(* www.hevs.ch Institut Systemes Industriels Project: HEVS Pack 2022 Author: Cedric Lenoir Date: 2024 August 30 This Function Block compute time statistics *)
FUNCTION_BLOCK FB_PackStatistic
  VAR_INPUT
    Enable : BOOL;
  END_VAR
  VAR_IN_OUT
    plcCurrentTime_s : UDINT;  (* E.g from PackTag.hevsPackTime.Local_date_time_seconds *)
    unitCurrentMode : E_PackModes;
    unitCurrentState : E_PackState;
    unitAdmin : HEVS_PackTag_Admin;
  END_VAR
  VAR_OUTPUT
    Active : BOOL;
  END_VAR
  VAR
    trigModeTimeCurrent : R_TRIG;  (* Detext State / Mode change *)
    trigStateTimeCurrent : R_TRIG;
    memCurrentMode : E_PackModes := E_PackModes.Invalid;
    memCurrentState : E_PackState := E_PackState.eUndefined;
    timeModeAtTrigger_s : UDINT;  (* Start time at trigger to compute current *)
    timeStateAtTrigger_s : UDINT;
    bProgramStarted : BOOL;
    timeProgramStarted_s : UDINT;
    getMemCumTimeMode : DINT;  (* Get Time In CumulativeTime for Mode and or state *)
    getMemCumTimeModeState : DINT;
  END_VAR

                  IF Enable THEN
	trigModeTimeCurrent(clk := (unitCurrentMode <> memCurrentMode));
	trigStateTimeCurrent(clk := (unitCurrentState <> memCurrentState));
	
	IF trigModeTimeCurrent.Q THEN
		timeModeAtTrigger_s := plcCurrentTime_s;
		memCurrentMode := unitCurrentMode;
		// Get Stored value to compute new cummulative time.
		getMemCumTimeMode := unitAdmin.CumulativeTime[0].ModeStateTimes[unitCurrentMode].Mode;
	END_IF
	
	IF trigStateTimeCurrent.Q THEN
		timeStateAtTrigger_s := plcCurrentTime_s;
		memCurrentState := unitCurrentState;
	END_IF
	
	// If mode or state changed
	IF trigModeTimeCurrent.Q  OR
	   trigStateTimeCurrent.Q THEN
	   getMemCumTimeModeState := unitAdmin.CumulativeTime[0].ModeStateTimes[unitCurrentMode].State[memCurrentState];
	END_IF
	
	IF NOT bProgramStarted THEN
		bProgramStarted := TRUE;
		timeProgramStarted_s := plcCurrentTime_s;
	END_IF
	
	unitAdmin.ModeTimeCurrent := UDINT_TO_DINT(plcCurrentTime_s - timeModeAtTrigger_s);
	
	unitAdmin.StateTimeCurrent := UDINT_TO_DINT(plcCurrentTime_s - timeStateAtTrigger_s);
	
	// Default for [*] time from start program
	// No retain, that is number of Sec since last restart.
	unitAdmin.CumulativeTime[0].AccTimeSinceReset := UDINT_TO_DINT(plcCurrentTime_s - timeProgramStarted_s);
	
	// Minimum protection in case of unitCurrentMode exceed 
	//	HEVS_PackTag_GVL.C_MAXMODSTATESTIMES
	IF unitCurrentMode <= HEVS_PackTag_GVL.C_MAXMODSTATESTIMES THEN
		// getMemCumTimeMode is set only at trigger change mode
		unitAdmin.CumulativeTime[0].ModeStateTimes[unitCurrentMode].Mode := getMemCumTimeMode + unitAdmin.ModeTimeCurrent;
	END_IF
	
	// Minimum protection in case of unitCurrentMode exceed 
	//	HEVS_PackTag_GVL.C_MAXMODSTATESTIMES
	// 	HEVS_PackTag_GVL.C_MAXSTATES
	IF unitCurrentMode <= HEVS_PackTag_GVL.C_MAXMODSTATESTIMES AND
	   unitCurrentState <= HEVS_PackTag_GVL.C_MAXSTATES        THEN
		// getMemCumTimeModeState is set only at trigger change of mode OR state 
		unitAdmin.CumulativeTime[0].ModeStateTimes[unitCurrentMode].State[unitCurrentState] := getMemCumTimeModeState +  unitAdmin.StateTimeCurrent;
	END_IF
	
	Active	:= FALSE;
ELSE
	
	Active	:= TRUE;
END_IF




                
END_FUNCTION_BLOCK

CONFIGURATION Application
  RESOURCE Application ON PLC
    {attribute 'qualified_only'}
    VAR_GLOBAL CONSTANT  (* HEVS_PackTag_GVL - List of PackTags based on ISA–TR88.00.02-2022 www.hevs.ch Institut Systemes Industriels / Power & Control Project: Automation Box CtrlX S3 Author: Romain Ferrari & Cedric Lenoir Date: 2024 July 31 !!!!!! The value of these constants have to be set by the user depending on the system it is implemented on. !!!!!!\\ *)
      C_MAXSTATES : INT := 17;  (* Max State number. 0 is invalid *)
      C_COMMAND_MAXREALPARAMS : INT := 8;
      C_COMMAND_MAXSTRINGPARAMS : INT := 2;  (* / *)
      C_COMMAND_MAXLREALPARAMS : INT := 8;  (* Used in one of the main PackTag branch of the HEVS_PackTag_V30 : Command *)
      C_COMMAND_MAXDINTPARAMS : INT := 8;
      C_COMMAND_MAXRECIPE : INT := 8;
      C_STATUS_MAXREALPARAMS : INT := 8;  (* / *)
      C_STATUS_MAXSTRINGPARAMS : INT := 2;  (* / *)
      C_STATUS_MAXLREALPARAMS : INT := 8;
      C_STATUS_MAXDINTPARAMS : INT := 8;  (* Used in one of the main PackTag branch of the HEVS_PackTag_V30 : Status *)
      C_STATUS_MAXRECIPE : INT := 8;
      C_STATUS_MAXSTACKLIGHT : INT := 8;
      C_ADMIN_MAXREALPARAMS : INT := 8;  (* / *)
      C_ADMIN_MAXSTRINGPARAMS : INT := 2;  (* / *)
      C_ADMIN_MAXLREALPARAMS : INT := 8;
      C_ADMIN_MAXDINTPARAMS : INT := 8;
      C_ADMIN_MAXALARMS : INT := 20;
      C_ADMIN_MAXHISTORYALARMS : INT := 20;
      C_ADMIN_MAXWARNINGS : INT := 20;
      C_ADMIN_MAXCUMULATIVETIMES : INT := 3;  (* Minimum is 0 for [0], Arbitrarily initialized to 3 *)
      C_ADMIN_MAXPRODUCTDATA : INT := 11;
      C_ADMIN_MAXDISABLEDSTATES : INT := 8;
      C_ADMIN_MAXMODESTRANSITION : INT := 8;  (* is absolutely limited by C_ADMIN_MAXMODESTRANSITIONPACK *)
      C_ADMIN_MAXMODESTRANSITIONPACK : INT := 31;  (* as Pack used DWORD and 0 is reserved, max is limited to 31 *)
      C_MAXMODSTATESTIMES : INT := 8;
      C_MAXREALVARIABLES : INT := 8;
      C_MAXSTRINGVARIABLES : INT := 8;
      C_MAXLREALVARIABLES : INT := 8;
      C_MAXDINTVARIABLES : INT := 8;  (* Used in lower branches of the HEVS_PackTag_V30 *)
      C_MAXREALINGREDIENTS : INT := 8;
      C_MAXSTRINGINGREDIENTS : INT := 8;
      C_MAXLREALINGREDIENTS : INT := 8;
      C_MAXDINTINGREDIENTS : INT := 8;
      hevs_min_packtag_v2022 : HEVS_Min_PackTag_V2022;
    END_VAR
    {attribute 'qualified_only'}
    VAR_GLOBAL  (* PackTag - www.hevs.ch Institut Systemes Industriels Project: HEVS Pack 2022 Author: Cedric Lenoir Date: 2024 August 29 Base GVL for HEVS Pack Tag File name should be PackTag *)
      Command : HEVS_PackTag_Command;
      Status : HEVS_PackTag_Status;
      Admin : HEVS_PackTag_Admin;
      hevsPackTime : HEVS_Time;  (* HEVS Time, needed for Alarms and Time in Pack Computed with PRG_GetTime_CtrlX or PRG_GetTime_TwinCAT or Your own system *)
      hevsUI : HEVS_PackTag_UI;  (* Help for interface and diagnostic HEVS Pack could be used without this Struct. Can be used with fbCmdBoolInterface Can be used with fbGetActualBoolState *)
      hevsPackAlarm_UI : HEVS_PackAlarm_UI;  (* Help for interface and diagnostic HEVS Pack could be used without this Struct. Can be used with program PRG_TestAlarm *)
    END_VAR
    {attribute 'qualified_only'}
    VAR_GLOBAL  (* GVL_Node - Some GVL to test var with NodeRED. Source: www.hevs.ch Author: Cedric Lenoir Date: 22 August 2024 *)
      readREAL : REAL;
      readDINT : DINT;
      readBOOL : BOOL;
      readString : STRING;
      writeREAL : REAL;
      writeDINT : DINT;
      writeBOOL : BOOL;
    END_VAR
    TASK MainTask(INTERVAL := T#4ms, PRIORITY := 30);
    PROGRAM PRG_GetTime_CtrlX WITH MainTask : PRG_GetTime_CtrlX;
    PROGRAM PLC_PACK WITH MainTask : PLC_PACK;
    PROGRAM PRG_TestAlarm WITH MainTask : PRG_TestAlarm;
    PROGRAM PRG_Sandbox WITH MainTask : PRG_Sandbox;
  END_RESOURCE
END_CONFIGURATION
